PROGRAM PRG_UpdateTemperatureControl
VAR
	tempControlMode				: EN_TempControlMode := EN_TempControlMode.TEMP_MODE_MANUAL;  
	
	loopCounter					: DINT := 0;

	(* Controller settings *)
	pwmPeriodinSec			: TIME := T#25S;
	pwmDutyCycle			: REAL := 0.0;	
	pwmOutputValveControl 	: FB_PWM;
	
	pidController			: FT_PIDWL;
	
	kp_heating				: REAL := 0.002;
	tv_heating				: REAL := 200;
	tn_heating				: REAL := 1800;
	
	kp_cooling				: REAL := 0.006;
	tv_cooling				: REAL := 200;
	tn_cooling				: REAL := 1800;

	kp_steri				: REAL := 0.0065;
	tv_steri				: REAL := 200;
	tn_steri				: REAL := 300;
	
	kp						: REAL := kp_heating;
	tv						: REAL := tv_heating;
	tn						: REAL := tn_heating;

	(* KD = KP*TV *)			
	(* KI = KP/TN *)
	
	errorTemp				: REAL := 0.0;
	pidReset				: BOOL := FALSE;
		
	evtSteriStart			: DetectEvent;
	evtSteriStop			: DetectEvent;
		
	evtTempControlStart		: DetectEvent;
	evtTempControlStop		: DetectEvent;
	
	windUpResetTimer		: TON;
	windUpResetTime			: TIME := T#30S;
	
	maxValveOnTimer		 	: TON;
	maxValveOnTime			: TIME := T#25S;	
	
	evtPidReset				: DetectEvent;
	(*
	myPwmBlock				: FB_PWM;
	pwmCycleTime			: TIME := T#2S;
	myPwmDutyCycle			: REAL := 0.5;
	*)
END_VAR

(* jacket temperature input *)
jacketTempC := INT_TO_REAL(jacketTempRaw)/32768.0*200.0 -50.0;
jacketTempK := jacketTempC + 273.15;
tOrpCurrent;

evtSteriStart(		newSignalValue := steriStart);
evtSteriStop(		newSignalValue := steriStop);
evtTempControlStart(newSignalValue := tempControlStart);
evtTempControlStop(	newSignalValue := tempControlStop);
evtPidReset( 		newSignalValue := pidReset);


IF evtSteriStart.eventDetected = TASTEVT_PositiveEdge THEN
	steriStart := FALSE;
	pumpOn := FALSE;
	pidController( RST:= TRUE );
	tempControlMode	:= EN_TempControlMode.TEMP_MODE_STERI;
	tempControlRunning := FALSE;
	steriRunning := TRUE;
	steriValve := FALSE;
	coldValve := FALSE;
	hotValve := FALSE;
	(* Set remaining steri temp *)
	remainingSteriTimeInMs := targetSteriTimeMinutes*60*1000; 
END_IF

IF evtTempControlStart.eventDetected = TASTEVT_PositiveEdge THEN
	tempControlStart := FALSE;
	pumpOn := FALSE;
	pidController( RST:= TRUE );
	tempControlMode	:= EN_TempControlMode.TEMP_MODE_HEATCOOL;
	tempControlRunning := TRUE;
	steriRunning := FALSE;
	steriValve := FALSE;
	coldValve := FALSE;
	hotValve := FALSE;
END_IF

IF 	evtSteriStop.eventDetected = TASTEVT_PositiveEdge OR
 	evtTempControlStop.eventDetected = TASTEVT_PositiveEdge 
THEN
	steriStop := FALSE;
	tempControlStop := FALSE;
	pumpOn := FALSE;
	pidController( RST:= TRUE );
	tempControlRunning := FALSE;
	steriRunning := FALSE;
	tempControlMode	:= EN_TempControlMode.TEMP_MODE_MANUAL;
	coldValve := FALSE;
	hotValve := FALSE;
	steriValve := FALSE;
	(* TODO: Reset Steri Timer *)
END_IF

CASE tempControlMode OF
	EN_TempControlMode.TEMP_MODE_MANUAL:
		pumpOn := FALSE;
		pidController( RST:= TRUE );
		
	EN_TempControlMode.TEMP_MODE_HEATCOOL:
	
		
		pumpOn := TRUE;
		(* errorTemp := targetControlTemp - currentMeanTemp; *)
		errorTemp := FUN_ComputeMovingSetPoint(currentTemp := currentMeanTemp, targetSetPoint := targetControlTemp) - currentMeanTemp;
		
		pidController(	IN:= errorTemp,
						KP:= kp,
						TN:= tn,
						TV:= tv,
						LIM_L:= -1.0,
						LIM_H:= 1.0,
						RST:= pidReset);
						
		(* pwmDutyCycle := ABS(pidController.Y); (* !! pwm block cannot handle negative inputs *) *)
		(* pwmDutyCycle := 0.05; *)
		
		
		pwmOutputValveControl(pwmCycleTime:=pwmPeriodinSec, pwmDutyCycle:=pwmDutyCycle);	
		
		
		IF pidController.Y > 0 THEN
			(* heating *)
			coldValve := FALSE;
			hotValve := pwmOutputValveControl.Q;
			kp := kp_heating;
			tv := tv_heating;
			tn := tn_heating;
			
		ELSE
			(* cooling *)
			coldValve := pwmOutputValveControl.Q;
			hotValve := FALSE;

			kp := kp_cooling;
			tv := tv_cooling;
			tn := tn_cooling;
		END_IF
		
	
	EN_TempControlMode.TEMP_MODE_STERI:
		pumpOn := FALSE;
		errorTemp := targetSteriTemp - currentMeanTemp;
		pidController(	IN:= errorTemp,
						KP:= kp_steri,
						TN:= tn_steri,
						TV:= tv_steri,
						LIM_L:= -1.0,
						LIM_H:= 1.0,
						RST:= pidReset);
						
		pwmDutyCycle := ABS(pidController.Y); (* !! pwm block cannot handle negative inputs *)
		
		pwmOutputValveControl(pwmCycleTime:=pwmPeriodinSec, pwmDutyCycle:=pwmDutyCycle);
				
		IF pidController.Y > 0 THEN
			(* heating *)
			coldValve := FALSE;
			steriValve := pwmOutputValveControl.Q;
		ELSE
			(* cooling *)
			(* coldValve := pwmOutputValveControl.Q; *)
			steriValve := FALSE;
		END_IF
		
		IF currentMeanTemp > (targetSteriTemp-0.5) THEN
			(* count down 10 ms each cycle *)
			remainingSteriTimeInMs := remainingSteriTimeInMs - 10;
			IF remainingSteriTimeInMs < 0 THEN
				tempControlMode := EN_TempControlMode.TEMP_MODE_MANUAL;
				steriValve := FALSE;
				coldValve := FALSE;
				steriStop := TRUE;
			END_IF
		END_IF		
		remainingSteriTimeMinutes := DINT_TO_REAL(remainingSteriTimeInMs)/(60.0*1000.0);
	
	
END_CASE

(*
maxValveOnTimer(IN:= (coldValve OR hotValve OR steriValve), PT:= maxValveOnTime);
IF maxValveOnTimer.Q THEN
	maxValveOnTimer(IN:=FALSE);
	countValveMaxTimeExceeded := countValveMaxTimeExceeded + 1;
	pidReset := TRUE;
	steriValve := FALSE;
	coldValve := FALSE;
	hotValve := FALSE;
END_IF
*)
(*
IF tempSafetyEnabled THEN
	IF (tPhLastReadingValid = FALSE AND tOrpLastReadingValid = FALSE) OR
		(currentMeanTemp > targetControlTemp + 0.5 OR currentMeanTemp < targetControlTemp - 0.5) THEN
		//tempControlMode := EN_TempControlMode.TEMP_MODE_MANUAL;
		pidReset := TRUE;
		countTempSpikes := countTempSpikes + 1;
		steriValve := FALSE;
		coldValve := FALSE;
		hotValve := FALSE;
	END_IF
END_IF
*)
 
IF evtPidReset.eventDetected = TASTEVT_PositiveEdge THEN
	pidReset := FALSE;
	pidController(RST:=TRUE);
	pidResetCounter := pidResetCounter + 1;
	steriValve := FALSE;
	coldValve := FALSE;
	hotValve := FALSE;
END_IF

END_PROGRAM

(* stored: Version 1.1.0.1, ProductVersion 3.1.4022.7
   POU PRG_UpdateTemperatureControl: Id {ef85cfaf-e33e-45d1-bc6c-ab2b3e926367}, SpecialFunc None *)
